(* Logix 5000 project; controller CI_CD_Example_Project vendor 1 type 14 code 196 rev 37.11; software revision 37.00 *)

TASK MainTask (continuous, watchdog 500 ms) : MainProgram

MODULES
   Local : vendor 1 type 14 code 196 (5069 0, rev 37.11)
END_MODULES

VAR_GLOBAL   (* controller tags *)
   Motor_Starter : BOOL;
   Start_Motor : BOOL;
   Stop_Motor : BOOL;
END_VAR

PROGRAM MainProgram   (* main routine MainRoutine *)
VAR
   E_Stop_Okay : BOOL;
   Master_Power_Safety : BOOL;
   Operator_Mode_Active : BOOL;
   Robot_Okay : BOOL;
   Safety_Scanner_Okay : BOOL;
END_VAR

ROUTINE MainRoutine   (* ladder *)
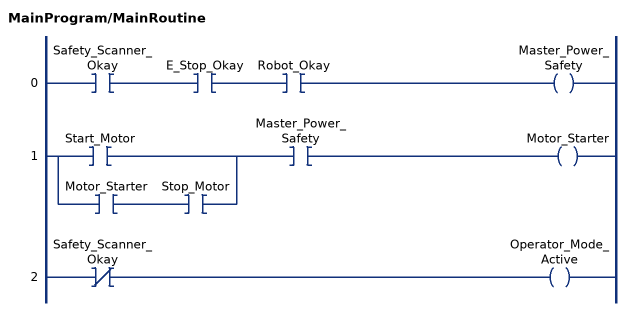
   0: XIC(Safety_Scanner_Okay)XIC(E_Stop_Okay)XIC(Robot_Okay)OTE(Master_Power_Safety);
   1: [XIC(Start_Motor) ,XIC(Motor_Starter) XIC(Stop_Motor) ]XIC(Master_Power_Safety)OTE(Motor_Starter);
   2: XIO(Safety_Scanner_Okay)OTE(Operator_Mode_Active);
END_ROUTINE
END_PROGRAM
